// TIA Portal V20 export
DATA_BLOCK "timer ON_DB"   // DB9
// stored: InstanceOfName timer ON, InstanceOfType FB
"timer ON"
   // VAR_OUTPUT
   //    second : Int;
   //    minutes : Int;
   //    hours : Real;
   //    days : Real;
   //    years : Real;
   // END_VAR
   // VAR
   //    P_TRIG : Bool;
   //    Timer_R : Bool;
   // END_VAR
BEGIN
END_DATA_BLOCK
